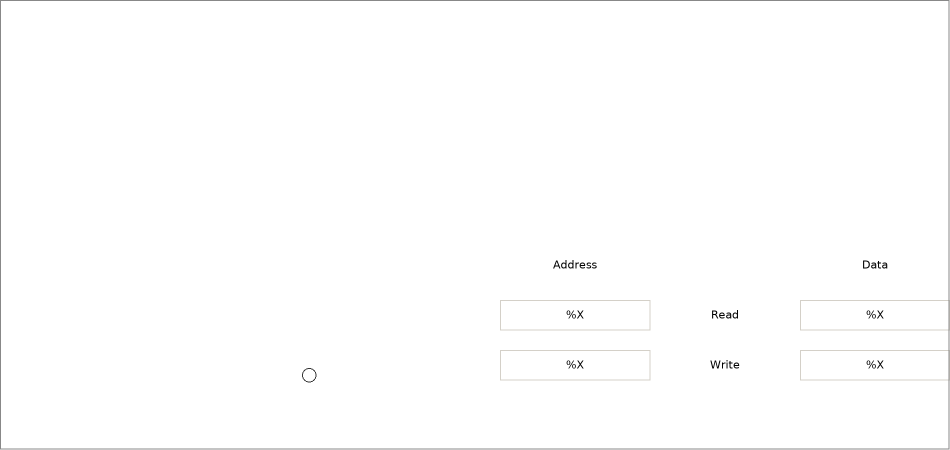
VISUALIZATION Visualization  // 950x450
    RadioButton (300,300 150x150), variable: MAIN.state
        Areas[0]: Text=Init
        Areas[1]: Text=ReadInputReg
        Areas[2]: Text=ReadReg
        Areas[3]: Text=WriteReg
    Textfield (500,300 150x30), "%X", text variable: MAIN.mbReadAddr
        OnMouseClick: write the text variable via Default, format %X
    Label (650,300 150x30), "Read"
    Label (500,250 150x30), "Address"
    Label (800,250 150x30), "Data"
    Textfield (800,300 150x30), "%X", text variable: MAIN.mbReadData
    Textfield (800,350 150x30), "%X", text variable: MAIN.mbWriteData
        OnMouseClick: write the text variable via Default
    Textfield (500,350 150x30), "%X", text variable: MAIN.mbWriteAddr
        OnMouseClick: write the text variable via Default, format %X
    Label (650,350 150x30), "Write"
END_VISUALIZATION

(* stored: Version 1.1.0.1, ProductVersion 3.1.4024.6
   Visu Visualization: Id {4f66a926-c9c2-48ee-9c5f-ba36a81e002c} *)
